(* PLC project EPEC_CU1.project, CODESYS V3.5 SP10 *)
(* stored: creationDateTime 2025-02-24T16:09:32.552285-06:00, modificationDateTime 2025-02-24T16:09:32.552285-06:00 *)

(* NOTE! NOTE! NOTE! NOTE! NOTE! NOTE! NOTE! NOTE! NOTE! NOTE! NOTE! This object is created by Epec MultiTool. User changes are overwritten when project is imported. Content: - EventCode channel IDs *)
{attribute 'qualified_only'}
{attribute 'strict'}
TYPE ChannelIDs : (Ch1 := 0, Ch2, Ch3, Ch4) BYTE;
END_TYPE

(* NOTE! NOTE! NOTE! NOTE! NOTE! NOTE! NOTE! NOTE! NOTE! NOTE! NOTE! This object is created by Epec MultiTool. User changes are overwritten when project is imported. Content: - EventCode device IDs *)
{attribute 'qualified_only'}
{attribute 'strict'}
TYPE DeviceIDs : (VoltageInput := 0, DigitalInput, CurrentInput, ParameterValidation) BYTE;
END_TYPE

TYPE IdentityObject : STRUCT
  VendorId : DWORD := 0;  (* Vendor ID *)
  ProductCode : DWORD := 0;  (* Product code *)
  Revision : DWORD := 0;  (* Revision number *)
  SerialNumber : DWORD := 0;  (* Serial number for control unit *)
END_STRUCT;
END_TYPE

VAR_GLOBAL CONSTANT  (* G_CONSTANTS - NOTE! NOTE! NOTE! NOTE! NOTE! NOTE! NOTE! NOTE! NOTE! NOTE! NOTE! This object is created by Epec MultiTool. User changes are overwritten when project is imported. Content: - Project specific constant definitions *)
  DIAG_TEMP_HIGH_LIMIT : DINT := 105;  (* Diagnostic limit constants *)
  DIAG_TEMP_LOW_LIMIT : DINT := -35;
  DIAG_TEMP_DELAY : UINT := 50;
  DIAG_SUPPLY_VOLTAGE_HIGH_LIMIT : DINT := 34000;
  DIAG_SUPPLY_VOLTAGE_LOW_LIMIT : DINT := 9000;
  DIAG_SUPPLY_VOLTAGE_DELAY : UINT := 95;
  DIAG_OUTPUT_GROUP1_HIGH_LIMIT : DINT := 34000;
  DIAG_OUTPUT_GROUP1_LOW_LIMIT : DINT := 9000;
  DIAG_OUTPUT_GROUP1_DELAY : UINT := 95;
  DIAG_5V_VAN_HIGH_LIMIT : DINT := 5250;
  DIAG_5V_VAN_LOW_LIMIT : DINT := 4750;
  DIAG_5V_VAN_DELAY : UINT := 50;
  DIAG_REF_DELAY : UINT := 50;
  DIAG_REF_TYPE_5V : BOOL := TRUE;  (* Reference output range selection [ TRUE = 5V, FALSE = 10V ] *)
  G_PARAMHANDLERKEYWORD : DWORD := 16#4EB1DA68;  (* Parameterhandler keyword *)
  G_PARAMETER_SAVE_STATUS_ERROR : BYTE := BYTE#16#00;
  G_PARAMETER_SAVE_STATUS_DONE : BYTE := BYTE#16#01;
  G_PARAMETER_SAVE_STATUS_IN_PROGRESS : BYTE := BYTE#16#FF;
  G_SAFE_PARAMETERS_AUTHENTICATED : BYTE := BYTE#1;
  G_SAFE_PARAMETERS_NOT_AUTHENTICATED : BYTE := BYTE#0;
END_VAR

{attribute 'qualified_only'}
VAR_GLOBAL  (* G_CAN - NOTE! NOTE! NOTE! NOTE! NOTE! NOTE! NOTE! NOTE! NOTE! NOTE! NOTE! This object is created by Epec MultiTool. User changes are overwritten when project is imported. Content: - CAN definitions *)
  Channel1 : EPEC_CANL2.Channel;
  Channel2 : EPEC_CANL2.Channel;
END_VAR

{attribute 'qualified_only'}
{attribute 'location' := '16#800'}
VAR_GLOBAL  (* G_Common *)
  ParHandler : EPEC_PH.ParameterHandler;  (* Parameterhandler. Utility library for ODSave. Library handles parameter image modification. *)
  ParameterArea : ARRAY[1..EPEC_HWD.LibParameters.G_PARAM_AREA_MAX_SIZE] OF BYTE;  (* Parameter image *)
  FastParHandler : EPEC_PH.ParameterHandler;
  FastParameterArea : ARRAY[1..EPEC_HWD.LibParameters.G_USER_VALUE_AREA_MAX_SIZE] OF BYTE;
  FastParameters : FastParameters;
  SaveFastParameters : BOOL := FALSE;
  ProjectKey : STRING(79) := '2JnCsjKPnmjYPqk';  (* Project key, used for validating the response code *)
END_VAR


{attribute 'qualified_only'}
{attribute 'location' := '16#800'}
VAR_GLOBAL  (* G_Logs *)
  ApplicationLog : EPEC_SERRLOG.ErrorLog;
  AppLogInitOK : BOOL;
END_VAR


{attribute 'qualified_only'}
{attribute 'location' := '16#800'}
VAR_GLOBAL  (* G_StatusFlags - NOTE! NOTE! NOTE! NOTE! NOTE! NOTE! NOTE! NOTE! NOTE! NOTE! NOTE! This object is created by Epec MultiTool. User changes are overwritten when project is imported. Content: - PLC_PRG status flags *)
  CANopenCan1NMTResetRequest : BOOL := FALSE;  (* Reset request flags tell if module is wanted to reset after current application cycle. *)
  CANopenCan2NMTResetRequest : BOOL := FALSE;
  SystemOk : BOOL := FALSE;
  CustomLEDControlEnable : BOOL := FALSE;  (* Flags to control the status LED from the application *)
  RedLED : BOOL := FALSE;
  GreenLED : BOOL := FALSE;
  BlueLED : BOOL := FALSE;
END_VAR

{attribute 'qualified_only'}
{attribute 'location' := '16#800'}
VAR_GLOBAL  (* G_SystemInfo - NOTE! NOTE! NOTE! NOTE! NOTE! NOTE! NOTE! NOTE! NOTE! NOTE! NOTE! This object is created by Epec MultiTool. User changes are overwritten when project is imported. Content: - System information common for all ODs. *)
  ProjectInfo : PROJECT_INFO;
  DeviceName : STRING(79);  (* 16#1008: Manufacturer device name *)
  HWVersion : STRING(79);  (* 16#1009: Manufacturer hardware version *)
  SWVersion : STRING(79);  (* 16#100A: Manufacturer software version *)
  Identity : IdentityObject;  (* 16#1018: Identity object *)
  ToolsVersion : ARRAY[1..1] OF DWORD;  (* 16#2030 Codesys version *)
  SoftwareInformation : ARRAY[1..10] OF STRING(79) := [''];  (* 16#2130 Software information Sub1: Application version Sub2: Additional version information Sub3: Reserved for future use Sub4: Reserved for future use Sub5: Reserved for future use Sub6: Reserved for future use Sub7: Reserved for future use Sub8: Reserved for future use Sub9: Reserved for future use Sub10: Reserved for future use *)
  CAN1_Comms : ARRAY[1..10] OF WORD := [10(0)];  (* 16#2150 CAN 1 Communication parameters Sub1: CODESYS communication enabled Sub2: CODESYS communication node-ID Sub3: Bit rate Sub4: Cable detection offset for CODESYS node-ID Sub5: Cable detection offset for PLCopen node-ID Sub6: Mask for cable detection pins Sub7: Reserved Sub8: Reserved Sub9: Reserved Sub10: PLCopen application node-ID in CAN1 *)
  CAN2_Comms : ARRAY[1..10] OF WORD := [10(0)];  (* 16#2151 CAN 2 Communication parameters Sub1: CODESYS communication enabled Sub2: CODESYS communication node-ID Sub3: Bit rate Sub4: Reserved Sub5: Reserved Sub6: Reserved Sub7: Reserved Sub8: Reserved Sub9: Reserved Sub10: PLCopen application node-ID in CAN2 *)
END_VAR

{attribute 'qualified_only'}
{attribute 'global_init_slot' := '49991'}
VAR_GLOBAL  (* G_CANopen_CAN1 - NOTE! NOTE! NOTE! NOTE! NOTE! NOTE! NOTE! NOTE! NOTE! NOTE! NOTE! This object is created by Epec MultiTool User changes are overwritten when project is imported Content - CANopen protocol variable definitions *)
  Device : EPEC_CANopen.Device;  (* CAN device *)
  OD : EPEC_CANopen.OD;  (* Object Dictionary data *)
  ODEntrys : ARRAY[1..70] OF EPEC_CANopen.ODEntry;
  Protocols : ARRAY[1..5] OF EPEC_CANopen.ProtocolEntry;  (* Protocol data *)
  HB : EPEC_CANopen.HBData;  (* Heartbeat producer/consumer protocol data *)
  HB_Handler : EPEC_CANopen.CANopenHB;  (* Heartbeat producer/consumer protocol handler *)
  NMT : EPEC_CANopen.NMTData;  (* NMT protocol data *)
  NMT_Handler : EPEC_CANopen.CANopenNMT;  (* NMT protocol handler *)
  SSDO : EPEC_CANopen.SSDOData;  (* SDO server protocol data *)
  SSDO_Handler : EPEC_CANopen.CANopenSDOServer;  (* SDO server protocol handler *)
  GFC : EPEC_CANopen.GFCData;  (* GFC protocol data *)
  GFC_Handler : EPEC_CANopen.CANopenGFC;  (* GFC protocol handler *)
  CSDOS : ARRAY[1..1] OF EPEC_CANopen.CANopenCSDO := [];  (* SDO client instances *)
  AppLogDomain : EPEC_CANopen.Domain;  (* 16#2171 Application log domain *)
  SaveAll : EPEC_ODSave.SaveODSaveAll;
  DeleteAll : EPEC_ODSave.SaveODDeleteAll;
  Initialize : EPEC_ODSave.SaveODInitialize;
  SaveData : ARRAY[0..3] OF EPEC_ODSave.SaveODSubIndexDescription := [(StartIndex := 16#1000, EndIndex := 16#FFFF, GroupNum := 1), (StartIndex := 16#1000, EndIndex := 16#1FFF, GroupNum := 1), (StartIndex := 16#2000, EndIndex := 16#FFFF, GroupNum := 1), (StartIndex := 16#0, EndIndex := 16#0, GroupNum := 1)];
  SaveSubData1010h : EPEC_ODSave.SaveODSubService;
END_VAR

{attribute 'qualified_only'}
{attribute 'location' := '16#800'}
{attribute 'global_init_slot' := '49990'}
VAR_GLOBAL  (* G_CANopen_CAN1_VAR - NOTE! NOTE! NOTE! NOTE! NOTE! NOTE! NOTE! NOTE! NOTE! NOTE! NOTE! This object is created by Epec MultiTool User changes are overwritten when project is imported Content - *)
  OD_Error : EPEC_CANopen.Errors := EPEC_CANopen.Errors.NotInitialized;
  ODSave_Error : EPEC_ODSave.SaveODErrors;
  Callback_Error : EPEC_CANopen.Errors := EPEC_CANopen.Errors.NotInitialized;
  ProtocolAdded : ARRAY[1..5] OF BOOL := [5(0)];
  HB_Error : EPEC_CANopen.Errors := EPEC_CANopen.Errors.NotInitialized;
  NMT_Error : EPEC_CANopen.Errors := EPEC_CANopen.Errors.NotInitialized;
  SSDO_Error : EPEC_CANopen.Errors := EPEC_CANopen.Errors.NotInitialized;
  GFC_Error : EPEC_CANopen.Errors := EPEC_CANopen.Errors.NotInitialized;
  GFC_Status : BYTE;  (* GFC status *)
  CSDO_Error : EPEC_CANopen.Errors := EPEC_CANopen.Errors.NotInitialized;
  SaveSigns1010 : ARRAY[0..3] OF DWORD;
END_VAR

{attribute 'qualified_only'}
{attribute 'location' := '16#800'}
VAR_GLOBAL  (* G_CAN1_VAR - NOTE! NOTE! NOTE! NOTE! NOTE! NOTE! NOTE! NOTE! NOTE! NOTE! NOTE! This object is created by Epec MultiTool User changes are overwritten when project is imported Content - CANopen OD index data *)
  DeviceType_Device1 : UDINT := 405;  (* 16#1000 Information about the device type *)
  ErrorReg_Device1 : USINT := 0;  (* 16#1001 Error information *)
  TPDO_DUMMY : BYTE := 0;  (* 16#2128 PDO Dummy Variable Index *)
  RPDO_DUMMY : BYTE := 0;  (* 16#2129 PDO Dummy Variable Index *)
  Parameter_CSV_unique_ID : UINT := 16#0000;  (* 16#2131 Parameter CSV unique ID *)
  ParameterSaveStatus : BYTE := 0;  (* 16#21FA Parameter save information *)
END_VAR

(* This PRG contains non safety-related code. The following attribute is autogenerated. Do not remove. *)
{attribute 'location' := '16#800'}
PROGRAM NVMemory
  VAR_INPUT
    i_Initialize : BOOL := TRUE;
  END_VAR
  VAR_OUTPUT
    o_InitReady : BOOL;
    o_InitError : BOOL;
    o_InputError : BOOL;
    o_ParameterBackupLoaded : BOOL;  (* Valid OD parameter backup image loaded during init. Note indication requires HWD lib 1.1.3.0. *)
    o_FastParameterBackupLoaded : BOOL;  (* Valid fast parameter backup image loaded during init. Note indication requires HWD lib 1.1.3.0. *)
    o_ODParameterError : EPEC_PH.ParamHandlerStatus := EPEC_PH.ParamHandlerStatus.NO_ERROR;
    o_FastParameterError : EPEC_PH.ParamHandlerStatus := EPEC_PH.ParamHandlerStatus.NO_ERROR;
    o_NVMemError : EPEC_SYSTEM.SYSTEM_ERROR_CODES := EPEC_SYSTEM.SYSTEM_ERROR_CODES.FW_ERR_OK;
    o_DM2Error : EPEC_PH.ParamHandlerStatus := EPEC_PH.ParamHandlerStatus.NO_ERROR;
    o_MachineTypeError : EPEC_PH.ParamHandlerStatus := EPEC_PH.ParamHandlerStatus.NO_ERROR;  (* Note indication requires HWD lib 1.1.5.0. *)
  END_VAR
  VAR
    parSaveBusy : BOOL := FALSE;
    parSaveDone : BOOL := FALSE;
    parSaveError : BOOL := FALSE;
    authenticated : BOOL := FALSE;
  END_VAR

            IF i_Initialize THEN
	EPEC_HWD.NVMem.SetParameterBackup(i_Enable := EPEC_HWD.LibParameters.G_PARAM_BACKUP_IN_USE);

	EPEC_HWD.NVMem.Init(
		i_NVMemoryIndex := 0,
		i_pParametersArea := ADR(G_Common.ParameterArea),
		i_ParameterAreaSize := SIZEOF(G_Common.ParameterArea),
		i_pParameterHandler := ADR(G_Common.ParHandler),
		i_pUserValuesArea := ADR(G_Common.FastParameterArea),
		i_UserValueAreaSize := SIZEOF(G_Common.FastParameterArea),
		i_pUserValueHandler := ADR(G_Common.FastParHandler),
		i_pUserValues := ADR(G_Common.FastParameters),
		i_UserValuesSize := SIZEOF(G_Common.FastParameters),
		i_pDM2Area := 0,
		i_DM2AreaSize := 0,
		i_pDM2Handler := 0,
		i_pMachineTypeArea := DWORD#0,
		i_MachineTypeAreaSize := UDINT#0,
		i_pMachineTypeHandler := DWORD#0,
		i_ParHandlerKeyword := G_CONSTANTS.G_PARAMHANDLERKEYWORD,
		o_InitReady => o_InitReady,
	);
	// Check if backup images were loaded during initialization
	IF o_InitReady THEN
		EPEC_HWD.NVMem.IsBackupLoaded(
			o_ParameterBackupLoaded => o_ParameterBackupLoaded,
			o_UserValueBackupLoaded => o_FastParameterBackupLoaded
		);
	END_IF
ELSE

	EPEC_HWD.NVMem(
		i_WriteParameters := G_Common.ParHandler.o_ParametersChanged,
		i_WriteUserValues := G_Common.SaveFastParameters,
		i_WriteDM2 := FALSE,
		i_WriteMachineType := FALSE,
		i_Authentication := authenticated,
		o_InitError => o_InitError,
		o_InputError => o_InputError,
		o_ParameterError => o_ODParameterError,
		o_UserValueError => o_FastParameterError,
		o_DM2Error => o_DM2Error,
		o_MachineTypeError => o_MachineTypeError,
		o_NVMemError => o_NVMemError,
		o_ParSaveBusy => parSaveBusy,
		o_ParSaveDone => parSaveDone,
		o_ParSaveError => parSaveError
	);

    (* Set parameter save status value *)
	IF parSaveBusy THEN
		G_CAN1_VAR.ParameterSaveStatus:= G_CONSTANTS.G_PARAMETER_SAVE_STATUS_IN_PROGRESS; 
	ELSIF parSaveDone THEN
		G_CAN1_VAR.ParameterSaveStatus:= G_CONSTANTS.G_PARAMETER_SAVE_STATUS_DONE; 
	ELSIF parSaveError THEN
		G_CAN1_VAR.ParameterSaveStatus:= G_CONSTANTS.G_PARAMETER_SAVE_STATUS_ERROR; 
	END_IF

	EPEC_SERRLOG.S_AddError_DWORD(i_ErrorCode:= ApplicationErrors.NVRAM_INIT, i_LibraryErrorCode:= BOOL_TO_DINT(o_InitError), i_Info1:= 0, i_Info2:= 0);
	EPEC_SERRLOG.S_AddError_DWORD(i_ErrorCode:= ApplicationErrors.NVRAM_INPUT, i_LibraryErrorCode:= BOOL_TO_DINT(o_InputError), i_Info1:= 0, i_Info2:= 0);
	EPEC_SERRLOG.S_AddError_DWORD(i_ErrorCode:= ApplicationErrors.NVRAM_FW, i_LibraryErrorCode:= o_NVMemError, i_Info1:= 0, i_Info2:= 0);
	EPEC_SERRLOG.S_AddError_DWORD(i_ErrorCode:= ApplicationErrors.NVRAM_OD, i_LibraryErrorCode:= INT_TO_DINT(o_ODParameterError), i_Info1:= 0, i_Info2:= 0);
	EPEC_SERRLOG.S_AddError_DWORD(i_ErrorCode:= ApplicationErrors.NVRAM_FASTPAR, i_LibraryErrorCode:= INT_TO_DINT(o_FastParameterError), i_Info1:= 0, i_Info2:= 0);
	EPEC_SERRLOG.S_AddError_DWORD(i_ErrorCode:= ApplicationErrors.NVRAM_MACHINETYPE, i_LibraryErrorCode:= INT_TO_DINT(o_MachineTypeError), i_Info1:= 0, i_Info2:= 0);


    (* User value save triggered, reset trigger *)
    G_Common.SaveFastParameters := FALSE;
END_IF
            
          
END_PROGRAM

(* Tool version : '8.1.9098.589' (MultiTool build version) Xml version : '1.0.10' (MultiTool xml file version) Control Unit : 'EPEC_CU1' (Name of the unit in MultiTool) Control Unit Type : 'EC44-020' (Type of the unit in MultiTool, including the functional version) CODESYS Profile : 'CODESYS V3.5 SP10' (CODESYS profile that was selected in MultiTool) Device Description Version: '3.5.13.67' (Device description version that was selected in MultiTool) Export Time : '24.02.2025 16:09.32' (Date and time when exported from MultiTool) Export Path : 'C:\Users\Pierre-Louis\Documents\02-UACH\1-Projets\1-Voltan\02-Réalisation\DEV\Projet_Voltan\Voltan_ECU\EPEC_CU1' (Path where MultiTool exported) Project File : 'C:\Users\Pierre-Louis\Documents\02-UACH\1-Projets\1-Voltan\02-Réalisation\DEV\Projet_Voltan\Voltan_ECU\Voltan_ECU.mtproject' (MultiTool project file name that was used) *)
{attribute 'location' := '16#800'}
PROGRAM PLC_PRG
  VAR_OUTPUT
    o_InitDone : BOOL := FALSE;
  END_VAR
  VAR
    ControlLED : EPEC_HWD.DiagnosticLED;
  END_VAR

            
// Initialize application log
IF NOT G_Logs.AppLogInitOK THEN
	G_Logs.AppLogInitOK := EPEC_SERRLOG.S_InitErrorLog(i_pErrorLog:= ADR(G_Logs.ApplicationLog));
END_IF

IF NOT o_InitDone AND G_Logs.AppLogInitOK THEN

    (* Code template non-safe FB initializations *)
    IF NOT Init_Entry.o_Ready THEN
        Init_Entry();
    ELSIF NOT Init_IO.o_Ready THEN
        Init_IO();
    ELSIF NOT EPEC_SHWD.S_EC44_Diagnostic.S_o_InitReady THEN
        EPEC_SHWD.S_EC44_Diagnostic.Init(
            S_i_SupplyVoltageHighLimit := G_CONSTANTS.DIAG_SUPPLY_VOLTAGE_HIGH_LIMIT,
            S_i_SupplyVoltageLowLimit := G_CONSTANTS.DIAG_SUPPLY_VOLTAGE_LOW_LIMIT,
            S_i_SupplyVoltageDiagDelay := G_CONSTANTS.DIAG_SUPPLY_VOLTAGE_DELAY,
            S_i_RefControlType5V := G_CONSTANTS.DIAG_REF_TYPE_5V,
            S_i_RefControlDiagDelay := G_CONSTANTS.DIAG_REF_DELAY,
            S_i_OutputGroup1HighVoltage := G_CONSTANTS.DIAG_OUTPUT_GROUP1_HIGH_LIMIT,
            S_i_OutputGroup1LowVoltage:= G_CONSTANTS.DIAG_OUTPUT_GROUP1_LOW_LIMIT,
            S_i_OutputGroup1DiagDelay:= G_CONSTANTS.DIAG_OUTPUT_GROUP1_DELAY,
            S_i_5VANHighVoltage:= G_CONSTANTS.DIAG_5V_VAN_HIGH_LIMIT,
            S_i_5VANLowVoltage:= G_CONSTANTS.DIAG_5V_VAN_LOW_LIMIT,
            S_i_5VANDiagDelay:= G_CONSTANTS.DIAG_5V_VAN_DELAY,
            S_i_TemperatureHighLimit:= G_CONSTANTS.DIAG_TEMP_HIGH_LIMIT,
            S_i_TemperatureLowLimit:= G_CONSTANTS.DIAG_TEMP_LOW_LIMIT,
            S_i_TemperatureDiagDelay:= G_CONSTANTS.DIAG_TEMP_DELAY);

    ELSIF NOT NVMemory.o_InitReady THEN
        NVMemory(i_Initialize:=TRUE);
	ELSIF NOT Inputs.o_InitReady THEN
		Inputs(i_Initialize:=TRUE);
	ELSIF NOT Init_CAN.o_Ready THEN
		Init_CAN();
	ELSIF NOT Init_CANopen_CAN1.o_Ready THEN
		Init_CANopen_CAN1();

    ELSE
        (* User non-safe initialization *)
        MainInit(o_MainInitReady=>o_InitDone);
    END_IF
ELSE
    (* Non-safe actions to execute before non-safe main program *)
	G_CAN.Channel1.CheckMessages();
	G_CAN.Channel2.CheckMessages();
	Inputs(i_Initialize:=FALSE);
	Handle_CANopen_CAN1();


    EPEC_SHWD.S_EC44_Diagnostic(
        i_RefChannel1  := Inputs.o_AI_REF_OUTPUT_MAIN_Diagnostic,
        i_SupplyVoltageInPin := Inputs.o_VIN_1_1_Diagnostic,
        i_SupplyBeforeSafetySwitch1 := Inputs.o_AI_POWER1_SUPPLY_Diagnostic,
        i_SupplyAfterSafetySwitch1  := Inputs.o_AI_POWER1_OUTPUT_Diagnostic,
        i_5VANChannel1 := Inputs.o_AI_5VAN_Diagnostic,
        i_PCBTemperatureChannel1 := Inputs.o_TEMP_PCB_MAIN_Diagnostic,
        i_PCBTemperatureChannel2 := Inputs.o_TEMP_PCB_RED_Diagnostic,
        i_MCUTemperature := Inputs.o_TEMP_MCU_Diagnostic,
        i_SBCTemperature := Inputs.o_AI_SBC_TEMP_Diagnostic
    );

	Handle_Diagnostic();

	// Read latest firmware errors to application log when FW is in error state
	IF EPEC_SHWD.S_EC44_Diagnostic.S_o_FWDiagnosticTaskStatus = EPEC_IODRV.DIAGNOSTIC_TASK_STATUS.EDiagnosticStatusError THEN
		Handle_Firmware_Errors(i_ReadErrors:= TRUE);
	END_IF


    (* User non-safe main program *)
    Main();

    (* Non-safe actions to execute after non-safe main program *)

    NVMemory(i_Initialize:=FALSE);

    (* Boot application if NMT reset requested *)
    IF G_StatusFlags.CANopenCan1NMTResetRequest OR G_StatusFlags.CANopenCan2NMTResetRequest THEN
        EPEC_SYSTEM.BOOT_APPLICATION_KILL_RTS();
    END_IF
END_IF

ControlLED(
    i_InitState := NOT PLC_PRG.o_Initdone,
    i_ApplicationInSafeState := NOT EPEC_SHWD.S_EC44_Diagnostic.S_o_OutputGroup1Control,
    i_SystemOk := G_StatusFlags.SystemOk,
    i_CustomLEDControl := G_StatusFlags.CustomLEDControlEnable,
    i_RedLED := G_StatusFlags.RedLED,
    i_GreenLED := G_StatusFlags.GreenLED,
    i_BlueLED := G_StatusFlags.BlueLED,
    o_Error =>
);


              
          
END_PROGRAM

(* NOTE! NOTE! NOTE! NOTE! NOTE! NOTE! NOTE! NOTE! NOTE! NOTE! NOTE! This object is created by Epec MultiTool User changes are overwritten when project is imported Content - Initialization of CAN channels This PRG contains non safety-related code. The following attribute is autogenerated. Do not remove. *)
{attribute 'location' := '16#800'}
PROGRAM Init_CAN
  VAR_OUTPUT
    o_Ready : BOOL := FALSE;
    o_Error : BOOL := FALSE;
    o_CAN1InitError : EPEC_CANVXD.ERROR := EPEC_CANVXD.ERROR.CHANNEL_NOT_INITIALIZED;
    o_CAN2InitError : EPEC_CANVXD.ERROR := EPEC_CANVXD.ERROR.CHANNEL_NOT_INITIALIZED;
  END_VAR

            o_CAN1InitError := G_CAN.Channel1.InitCAN(i_Channel := 0, i_BitRate := G_SystemInfo.CAN1_Comms[3], i_Flags := 0);
o_CAN2InitError := G_CAN.Channel2.InitCAN(i_Channel := 1, i_BitRate := EPEC_CANVXD.BITRATE_250K, i_Flags := 0);

IF EPEC_CANVXD.ERROR.NO_ERROR = o_CAN1InitError AND
	EPEC_CANVXD.ERROR.NO_ERROR = o_CAN2InitError THEN
	o_Error := FALSE;
ELSE
	o_Error := TRUE;

	EPEC_SERRLOG.S_AddError_DWORD(i_ErrorCode:= ApplicationErrors.CAN_INIT, i_LibraryErrorCode:= INT_TO_DINT(o_CAN1InitError), i_Info1:= 0, i_Info2:= 1);
	EPEC_SERRLOG.S_AddError_DWORD(i_ErrorCode:= ApplicationErrors.CAN_INIT, i_LibraryErrorCode:= INT_TO_DINT(o_CAN2InitError), i_Info1:= 0, i_Info2:= 2);
END_IF

o_Ready := TRUE;

          
END_PROGRAM

(* NOTE! NOTE! NOTE! NOTE! NOTE! NOTE! NOTE! NOTE! NOTE! NOTE! NOTE! This object is created by Epec MultiTool User changes are overwritten when project is imported Content - Set system information common for all ODs. This PRG contains non safety-related code. The following attribute is autogenerated. Do not remove. *)
{attribute 'location' := '16#800'}
PROGRAM Init_Entry
  VAR_OUTPUT
    o_Ready : BOOL;
  END_VAR
  VAR
    Can2NodeId : WORD;
    Can2PLCopenNodeId : WORD;
    Can2BitRate : WORD;
    ReadBytes : DWORD;
    RandomNumber : UDINT;
    SystemParameters : EPEC_HW.SystemParameters;
  END_VAR

            SystemParameters.ReadData();

/// 16#1008: Manufacturer device name
EPEC_SYSTEM.SystemParametersRead (16#1008,0,79,ADR(G_SystemInfo.DeviceName),ADR(ReadBytes));
 /// 16#1009: Manufacturer hardware version
EPEC_SYSTEM.SystemParametersRead (16#1009,0,79,ADR(G_SystemInfo.HWVersion),ADR(ReadBytes));
/// 16#100A: Manufacturer software version
G_SystemInfo.SWVersion := SystemParameters.o_SoftwareVersion;
/// 16#1018: Identity object 
G_SystemInfo.Identity.VendorId := SystemParameters.o_VendorId;          /// Vendor ID
G_SystemInfo.Identity.ProductCode := SystemParameters.o_ProductCode;    /// Product code
G_SystemInfo.Identity.Revision := SystemParameters.o_RevisionNumber;    /// Revision number
G_SystemInfo.Identity.SerialNumber := SystemParameters.o_SerialNumber;  /// Serial number for control unit
/// 16#2030 Codesys version
G_SystemInfo.ToolsVersion[1] := DWORD#50659328;
/// 16#2150 CAN 1 Communication parameters
G_SystemInfo.CAN1_Comms := SystemParameters.i_CAN1;

/// Read parameters for CAN2 from firmware
EPEC_SYSTEM.SystemParametersRead (16#2151,2,2,ADR(Can2NodeId),ADR(ReadBytes));
EPEC_SYSTEM.SystemParametersRead (16#2151,3,2,ADR(Can2BitRate),ADR(ReadBytes));
EPEC_SYSTEM.SystemParametersRead (16#2151,10,2,ADR(Can2PLCopenNodeId),ADR(ReadBytes));

/// Set variables to communication arrays 
G_SystemInfo.CAN2_Comms[2] := Can2NodeId;
G_SystemInfo.CAN2_Comms[3] := Can2BitRate;
G_SystemInfo.CAN2_Comms[10] := Can2PLCopenNodeId;

o_Ready:= TRUE;

          
END_PROGRAM

(* NOTE! NOTE! NOTE! NOTE! NOTE! NOTE! NOTE! NOTE! NOTE! NOTE! NOTE! This object is created by Epec MultiTool User changes are overwritten when project is imported Content - Non-safe system status update This PRG contains non safety-related code. The following attribute is autogenerated. Do not remove. *)
{attribute 'location' := '16#800'}
PROGRAM Handle_Diagnostic

            (* System Ok conditions *)
G_StatusFlags.SystemOk:=
		EPEC_SHWD.S_EC44_Diagnostic.S_o_DiagStatusOk AND			(* System diagnostic ok *)
		NOT Init_CAN.o_Error AND			(* No errors in bus init *)
		NOT Init_CANopen_CAN1.o_Error;


// Check HW diagnostic errors when diagnostic is enabled
IF EPEC_SHWD.S_EC44_Diagnostic.S_o_Running AND NOT EPEC_SHWD.S_EC44_Diagnostic.S_o_DiagStatusOk THEN
	EPEC_SERRLOG.S_AddError_DWORD(
		i_ErrorCode := ApplicationErrors.HW_DIAGNOSTIC_FAULT,
		i_LibraryErrorCode := EPEC_SERRLOG.LibConstants.G_ErrorNA,
		i_Info1 := 0,
		i_Info2 := 0);

	// output group 1
	EPEC_SERRLOG.S_AddError_BYTE(
		i_ErrorCode := ApplicationErrors.HW_DIAG_OUT_PWR_GRP_1,
		i_LibraryErrorCode := EPEC_SHWD.S_EC44_Diagnostic.o_OutputGroup1Control_EC.EventID,
		i_Info1 := EPEC_SHWD.S_EC44_Diagnostic.o_OutputGroup1Control_EC.FunctionID,
		i_Info2 := EPEC_SHWD.S_EC44_Diagnostic.o_OutputGroup1Control_EC.DeviceID,
		i_Info3 := EPEC_SHWD.S_EC44_Diagnostic.o_OutputGroup1Control_EC.ChannelID,
		i_Info4 := 0,
		i_Info5 := 0,
		i_Info6 := 0,
		i_Info7 := 0,
		i_Info8 := 0);

	// REF output
	EPEC_SERRLOG.S_AddError_BYTE(
		i_ErrorCode := ApplicationErrors.HW_DIAG_OUT_REF_1,
		i_LibraryErrorCode := EPEC_SHWD.S_EC44_Diagnostic.o_RefControl_EC.EventID,
		i_Info1 := EPEC_SHWD.S_EC44_Diagnostic.o_RefControl_EC.FunctionID,
		i_Info2 := EPEC_SHWD.S_EC44_Diagnostic.o_RefControl_EC.DeviceID,
		i_Info3 := EPEC_SHWD.S_EC44_Diagnostic.o_RefControl_EC.ChannelID,
		i_Info4 := 0,
		i_Info5 := 0,
		i_Info6 := 0,
		i_Info7 := 0,
		i_Info8 := 0);

	// supply voltage
	EPEC_SERRLOG.S_AddError_BYTE(
		i_ErrorCode := ApplicationErrors.HW_DIAG_IN_SUPPLY,
		i_LibraryErrorCode := EPEC_SHWD.S_EC44_Diagnostic.o_SupplyVoltag_EC.EventID,
		i_Info1 := EPEC_SHWD.S_EC44_Diagnostic.o_SupplyVoltag_EC.FunctionID,
		i_Info2 := EPEC_SHWD.S_EC44_Diagnostic.o_SupplyVoltag_EC.DeviceID,
		i_Info3 := EPEC_SHWD.S_EC44_Diagnostic.o_SupplyVoltag_EC.ChannelID,
		i_Info4 := 0,
		i_Info5 := 0,
		i_Info6 := 0,
		i_Info7 := 0,
		i_Info8 := 0);

	// 5VAN
	EPEC_SERRLOG.S_AddError_BYTE(
		i_ErrorCode := ApplicationErrors.HW_DIAG_IN_5VAN,
		i_LibraryErrorCode := EPEC_SHWD.S_EC44_Diagnostic.o_5VAN_EC.EventID,
		i_Info1 := EPEC_SHWD.S_EC44_Diagnostic.o_5VAN_EC.FunctionID,
		i_Info2 := EPEC_SHWD.S_EC44_Diagnostic.o_5VAN_EC.DeviceID,
		i_Info3 := EPEC_SHWD.S_EC44_Diagnostic.o_5VAN_EC.ChannelID,
		i_Info4 := 0,
		i_Info5 := 0,
		i_Info6 := 0,
		i_Info7 := 0,
		i_Info8 := 0);

	// MCU temperature
	EPEC_SERRLOG.S_AddError_BYTE(
		i_ErrorCode := ApplicationErrors.HW_DIAG_IN_MCU_TEMP,
		i_LibraryErrorCode := EPEC_SHWD.S_EC44_Diagnostic.o_MCUTemperatureEC.EventID,
		i_Info1 := EPEC_SHWD.S_EC44_Diagnostic.o_MCUTemperatureEC.FunctionID,
		i_Info2 := EPEC_SHWD.S_EC44_Diagnostic.o_MCUTemperatureEC.DeviceID,
		i_Info3 := EPEC_SHWD.S_EC44_Diagnostic.o_MCUTemperatureEC.ChannelID,
		i_Info4 := 0,
		i_Info5 := 0,
		i_Info6 := 0,
		i_Info7 := 0,
		i_Info8 := 0);

	// SBC temperature
	EPEC_SERRLOG.S_AddError_BYTE(
		i_ErrorCode := ApplicationErrors.HW_DIAG_IN_SBC_TEMP,
		i_LibraryErrorCode := EPEC_SHWD.S_EC44_Diagnostic.o_SBCTemperatureEC.EventID,
		i_Info1 := EPEC_SHWD.S_EC44_Diagnostic.o_SBCTemperatureEC.FunctionID,
		i_Info2 := EPEC_SHWD.S_EC44_Diagnostic.o_SBCTemperatureEC.DeviceID,
		i_Info3 := EPEC_SHWD.S_EC44_Diagnostic.o_SBCTemperatureEC.ChannelID,
		i_Info4 := 0,
		i_Info5 := 0,
		i_Info6 := 0,
		i_Info7 := 0,
		i_Info8 := 0);

	// PCB temperature 1
	EPEC_SERRLOG.S_AddError_BYTE(
		i_ErrorCode := ApplicationErrors.HW_DIAG_IN_PCB_TEMP_1,
		i_LibraryErrorCode := EPEC_SHWD.S_EC44_Diagnostic.o_PCBTemperatureCh1_EC.EventID,
		i_Info1 := EPEC_SHWD.S_EC44_Diagnostic.o_PCBTemperatureCh1_EC.FunctionID,
		i_Info2 := EPEC_SHWD.S_EC44_Diagnostic.o_PCBTemperatureCh1_EC.DeviceID,
		i_Info3 := EPEC_SHWD.S_EC44_Diagnostic.o_PCBTemperatureCh1_EC.ChannelID,
		i_Info4 := 0,
		i_Info5 := 0,
		i_Info6 := 0,
		i_Info7 := 0,
		i_Info8 := 0);

	// PCB temperature 2
	EPEC_SERRLOG.S_AddError_BYTE(
		i_ErrorCode := ApplicationErrors.HW_DIAG_IN_PCB_TEMP_2,
		i_LibraryErrorCode := EPEC_SHWD.S_EC44_Diagnostic.o_PCBTemperatureCh2_EC.EventID,
		i_Info1 := EPEC_SHWD.S_EC44_Diagnostic.o_PCBTemperatureCh2_EC.FunctionID,
		i_Info2 := EPEC_SHWD.S_EC44_Diagnostic.o_PCBTemperatureCh2_EC.DeviceID,
		i_Info3 := EPEC_SHWD.S_EC44_Diagnostic.o_PCBTemperatureCh2_EC.ChannelID,
		i_Info4 := 0,
		i_Info5 := 0,
		i_Info6 := 0,
		i_Info7 := 0,
		i_Info8 := 0);

END_IF



          
END_PROGRAM

(* NOTE! NOTE! NOTE! NOTE! NOTE! NOTE! NOTE! NOTE! NOTE! NOTE! NOTE! This object is created by Epec MultiTool User changes are overwritten when project is imported Content - Reads firmware error codes to application error log This PRG contains non safety-related code. The following attribute is autogenerated. Do not remove. *)
{attribute 'location' := '16#800'}
PROGRAM Handle_Firmware_Errors
  VAR_INPUT
    i_ReadErrors : BOOL;
  END_VAR
  VAR
    readErrorsOld : BOOL;
    fw_entries : ARRAY [1..EPEC_SERRLOG.LibParameters.G_ERROR_LOG_MAX_LINES] OF EPEC_SYSTEM.SystemLogEntry;
    return_code : EPEC_SYSTEM.SYSTEM_ERROR_CODES;
    lines_found : UDINT;
    i : UDINT;
    previous_time : UDINT;
    boot_detected : BOOL;
    fw_log_startupid : UDINT := UDINT#0;
    fw_log_startupid_exist : BOOL := FALSE;
    fw_log_startupid_size : DWORD;
  END_VAR

            IF i_ReadErrors AND NOT readErrorsOld THEN
	// Read FW log startup id value, if supported by FW
	return_code := EPEC_SYSTEM.SystemParametersRead(i_Index:=16#2039, i_SubIndex:=2, i_pBufferSize:=SIZEOF(fw_log_startupid), i_pBuffer:=ADR(fw_log_startupid), i_pNbrOfReadByte:=ADR(fw_log_startupid_size));

	// Check if read was success
	IF return_code = EPEC_SYSTEM.SYSTEM_ERROR_CODES.FW_ERR_OK THEN
		fw_log_startupid_exist := TRUE;
	ELSE
		fw_log_startupid_exist := FALSE;
	END_IF

	// Read firmware errors
	return_code:= EPEC_SYSTEM.GetFWLogTail(
		i_Count:= EPEC_SERRLOG.LibParameters.G_ERROR_LOG_MAX_LINES,
		i_logEntryArray:= ADR(fw_entries),
		o_Found => lines_found
	);

	IF return_code = EPEC_SYSTEM.SYSTEM_ERROR_CODES.FW_ERR_OK AND lines_found > UDINT#0 THEN
		// Check if startup id is supported by FW
		IF fw_log_startupid_exist THEN
			// Add errors from buffer until startup id is found 
			FOR i:= 1 TO EPEC_SERRLOG.LibParameters.G_ERROR_LOG_MAX_LINES DO
				IF i <= lines_found AND fw_entries[i].Identifier >= fw_log_startupid THEN
					S_AddError_DWORD(
						i_ErrorCode:= ApplicationErrors.FW_ERROR,
						i_LibraryErrorCode:= fw_entries[i].Error,
						i_Info1:= fw_entries[i].Info,
						i_Info2:= fw_entries[i].Identifier);
				END_IF
			END_FOR
		ELSE
			// Add first error
			S_AddError_DWORD(
				i_ErrorCode:= ApplicationErrors.FW_ERROR,
				i_LibraryErrorCode:= fw_entries[1].Error,
				i_Info1:= fw_entries[1].Info,
				i_Info2:= fw_entries[1].Identifier);

			previous_time:= fw_entries[1].Timestamp;
			boot_detected:= FALSE;

			// Add errors until timestamp rollover is detected
			FOR i:= 2 TO EPEC_SERRLOG.LibParameters.G_ERROR_LOG_MAX_LINES DO
				IF i <= lines_found AND fw_entries[i].Timestamp <= previous_time AND NOT boot_detected THEN
					S_AddError_DWORD(
						i_ErrorCode:= ApplicationErrors.FW_ERROR,
						i_LibraryErrorCode:= fw_entries[i].Error,
						i_Info1:= fw_entries[i].Info,
						i_Info2:= fw_entries[i].Identifier);

					previous_time:= fw_entries[i].Timestamp;

				ELSIF fw_entries[i].Timestamp > previous_time THEN
					boot_detected := TRUE;
				END_IF
			END_FOR
		END_IF
	END_IF
END_IF
readErrorsOld:= i_ReadErrors;

          
END_PROGRAM

(* NOTE! NOTE! NOTE! NOTE! NOTE! NOTE! NOTE! NOTE! NOTE! NOTE! NOTE! This object is created by Epec MultiTool User changes are overwritten when project is imported Content - CANopen initialization - Includes Init_CANopen_OD1 - CANopen data update This PRG contains non safety-related code. The following attribute is autogenerated. Do not remove. *)
{attribute 'location' := '16#800'}
PROGRAM Init_CANopen_CAN1
  VAR_OUTPUT
    o_Ready : BOOL := FALSE;
    o_Error : BOOL := FALSE;
  END_VAR

            G_CANopen_CAN1.Device.itfCanChannel:=G_CAN.Channel1; (*Connect device to can channel*)
G_CANopen_CAN1.Device.NodeID := BYTE#1;
G_CANopen_CAN1.NMT.NmtState:=EPEC_CANopen.NMTState.BootUp; (* Set NMT status to BOOTUP *)

(*Initialize OD's data structures*)
G_CANopen_CAN1.OD.EntryCount:=SIZEOF(G_CANopen_CAN1.ODEntrys)/SIZEOF(G_CANopen_CAN1.ODEntrys[1]); (*Max entries of given OD(CANopenDeviceODEntrys array)*)
G_CANopen_CAN1.OD.InOrder:=FALSE; (*OD isn't in order*)
G_CANopen_CAN1.OD.NextFree:=0; (*OD does not have any entries yet*)
G_CANopen_CAN1.OD.pODEntry:=ADR(G_CANopen_CAN1.ODEntrys); (*Pointer to OD array*)

(*Define NMT protocol*)
G_CANopen_CAN1.Protocols[1].Protocol:=EPEC_CANopen.ProtocolType.NMT;
G_CANopen_CAN1.Protocols[1].pData:=ADR(G_CANopen_CAN1.NMT);
G_CANopen_CAN1.Protocols[1].itfProtocol:=G_CANopen_CAN1.NMT_Handler;
G_CANopen_CAN1.Protocols[1].pError:=ADR(G_CANopen_CAN1_VAR.NMT_Error);
G_CANopen_CAN1_VAR.ProtocolAdded[1] := CANopenDeviceAddProtocol( (* Add to protocol stack *)
	i_pDevice:=ADR(G_CANopen_CAN1.Device),
	i_pProtocol:=ADR(G_CANopen_CAN1.Protocols[1]),
);

(*Initialize NMT protocol*)
IF G_CANopen_CAN1_VAR.ProtocolAdded[1] THEN
	G_CANopen_CAN1.NMT_Handler.Init(
		i_pDevice := ADR(G_CANopen_CAN1.Device),
		i_ThisIsMaster := FALSE,
		i_StartInterval :=  1000,
		i_pMonitoredNodes := 0,
		i_NumberOfNodes := 0,
		i_SimultaneousSlaveConfiguration := FALSE,
		o_Error => G_CANopen_CAN1_VAR.NMT_Error
	);
ELSE
	G_CANopen_CAN1_VAR.NMT_Error := EPEC_CANopen.Errors.ProtocolDataMissing;
END_IF

(*Define OD protocol*)
G_CANopen_CAN1.Protocols[2].Protocol:=EPEC_CANopen.ProtocolType.OD;
G_CANopen_CAN1.Protocols[2].pData:=ADR(G_CANopen_CAN1.OD);
G_CANopen_CAN1.Protocols[2].pError:=ADR(G_CANopen_CAN1_VAR.OD_Error);
G_CANopen_CAN1_VAR.ProtocolAdded[2] := CANopenDeviceAddProtocol( (* Add to protocol stack *)
	i_pDevice:=ADR(G_CANopen_CAN1.Device),
	i_pProtocol:=ADR(G_CANopen_CAN1.Protocols[2]),
);
IF NOT G_CANopen_CAN1_VAR.ProtocolAdded[2] THEN
	G_CANopen_CAN1_VAR.OD_Error := EPEC_CANopen.Errors.ProtocolDataMissing;
END_IF

(*Define HB protocol
- Uses NMT and OD protocol data, thus need to be defined after them.
*)
G_CANopen_CAN1.HB.HeartBeat.PT := T#200MS; (* HB producer time *)

G_CANopen_CAN1.Protocols[3].Protocol:=EPEC_CANopen.ProtocolType.HB;
G_CANopen_CAN1.Protocols[3].pData:=ADR(G_CANopen_CAN1.HB);
G_CANopen_CAN1.Protocols[3].itfProtocol:=G_CANopen_CAN1.HB_Handler;
G_CANopen_CAN1.Protocols[3].pError:=ADR(G_CANopen_CAN1_VAR.HB_Error);
G_CANopen_CAN1_VAR.ProtocolAdded[3] := CANopenDeviceAddProtocol( (* Add to protocol stack *)
	i_pDevice:=ADR(G_CANopen_CAN1.Device),
	i_pProtocol:=ADR(G_CANopen_CAN1.Protocols[3]),
);

(* Initialize HB protocol *)
IF G_CANopen_CAN1_VAR.ProtocolAdded[3] THEN

	(* Add monitored nodes *)
	G_CANopen_CAN1.HB_Handler.Init(
		i_pDevice := ADR(G_CANopen_CAN1.Device),
		o_Error => G_CANopen_CAN1_VAR.HB_Error
	);
ELSE
	G_CANopen_CAN1_VAR.HB_Error := EPEC_CANopen.Errors.ProtocolDataMissing;
END_IF

(*Define SSDO protocol*)
G_CANopen_CAN1.Protocols[4].Protocol:=EPEC_CANopen.ProtocolType.SSDO;
G_CANopen_CAN1.Protocols[4].pData:=ADR(G_CANopen_CAN1.SSDO);
G_CANopen_CAN1.Protocols[4].itfProtocol:=G_CANopen_CAN1.SSDO_Handler;
G_CANopen_CAN1.Protocols[4].pError:=ADR(G_CANopen_CAN1_VAR.SSDO_Error);
G_CANopen_CAN1_VAR.ProtocolAdded[4] := CANopenDeviceAddProtocol( (* Add to protocol stack *)
	i_pDevice:=ADR(G_CANopen_CAN1.Device),
	i_pProtocol:=ADR(G_CANopen_CAN1.Protocols[4])
);
IF G_CANopen_CAN1_VAR.ProtocolAdded[4] THEN
	G_CANopen_CAN1.SSDO_Handler.Init(
		i_pDevice := ADR(G_CANopen_CAN1.Device),
		o_Error => G_CANopen_CAN1_VAR.SSDO_Error
	);
ELSE
	G_CANopen_CAN1_VAR.SSDO_Error := EPEC_CANopen.Errors.ProtocolDataMissing;
END_IF

(*Define GFC protocol*)
G_CANopen_CAN1.Protocols[5].Protocol:=EPEC_CANopen.ProtocolType.GFC;
G_CANopen_CAN1.Protocols[5].pData:=ADR(G_CANopen_CAN1.GFC);
G_CANopen_CAN1.Protocols[5].itfProtocol:=G_CANopen_CAN1.GFC_Handler;
G_CANopen_CAN1.Protocols[5].pError:=ADR(G_CANopen_CAN1_VAR.GFC_Error);
G_CANopen_CAN1_VAR.ProtocolAdded[5] := CANopenDeviceAddProtocol(  (* Add to protocol stack *)
	i_pDevice:=ADR(G_CANopen_CAN1.Device),
	i_pProtocol:=ADR(G_CANopen_CAN1.Protocols[5])
);
IF G_CANopen_CAN1_VAR.ProtocolAdded[5] THEN
	G_CANopen_CAN1.GFC_Handler.Init(
		i_pDevice := ADR(G_CANopen_CAN1.Device),
		i_pStatus:=ADR(G_CANopen_CAN1_VAR.GFC_Status),
		o_Error => G_CANopen_CAN1_VAR.GFC_Error
	);
ELSE
	G_CANopen_CAN1_VAR.GFC_Error := EPEC_CANopen.Errors.ProtocolDataMissing;
END_IF

(* Init CSDO instance array for bus *)
EPEC_CANopen.CANopenSDOManager.Init(
	i_pDevice:=ADR(G_CANopen_CAN1.Device),
	i_pCsdoArrayStart:=ADR(G_CANopen_CAN1.CSDOS),
	i_CsdoArraySize:=SIZEOF(G_CANopen_CAN1.CSDOS)/SIZEOF(G_CANopen_CAN1.CSDOS[1]),
	o_Error=>G_CANopen_CAN1_VAR.CSDO_Error
);

(* Add index data to OD *)
Init_CANopen_OD1(); (* Must be done before initing PDOs and SRDOs. *)

(*Initialize OD save*)
G_CANopen_CAN1.SaveAll.Init(i_pParamHandler:=ADR(G_Common.ParHandler));
G_CANopen_CAN1.DeleteAll.Init(i_pParamHandler:=ADR(G_Common.ParHandler));
G_CANopen_CAN1.SaveSubData1010h.pSaveSigns := ADR(G_CANopen_CAN1_VAR.SaveSigns1010[0]);
G_CANopen_CAN1.SaveSubData1010h.NumOfEntrys := 4;
G_CANopen_CAN1.SaveSubData1010h.pSaveIndexData := ADR(G_CANopen_CAN1.SaveData[0]);
G_CANopen_CAN1.SaveData[3].itfSaveAll := G_CANopen_CAN1.SaveAll;
G_CANopen_CAN1.SaveData[3].itfDeleteAll := G_CANopen_CAN1.DeleteAll;
G_CANopen_CAN1.OD.pAdditionalData := ADR(G_CANopen_CAN1.SaveSubData1010h);

IF G_CANopen_CAN1_VAR.OD_Error = EPEC_CANopen.Errors.NoError THEN
	G_CANopen_CAN1.Initialize(i_pOD:=ADR(G_CANopen_CAN1.OD), i_pParamHandler:=ADR(G_Common.ParHandler), o_Error => G_CANopen_CAN1_VAR.ODSave_Error);
END_IF

(* Check all protocol init status flags *)
IF G_CANopen_CAN1_VAR.NMT_Error = EPEC_CANopen.Errors.NoError AND
	G_CANopen_CAN1_VAR.SSDO_Error = EPEC_CANopen.Errors.NoError AND
	G_CANopen_CAN1_VAR.OD_Error = EPEC_CANopen.Errors.NoError AND
	G_CANopen_CAN1_VAR.HB_Error = EPEC_CANopen.Errors.NoError AND
	G_CANopen_CAN1_VAR.CSDO_Error = EPEC_CANopen.Errors.NoError AND
	G_CANopen_CAN1_VAR.GFC_Error = EPEC_CANopen.Errors.NoError
THEN
	o_Error := FALSE; (* No errors in protocol inits *)
ELSE
	o_Error := TRUE;

	EPEC_SERRLOG.S_AddError_DWORD(i_ErrorCode:= ApplicationErrors.CANOPEN_INIT_NMT, i_LibraryErrorCode:= INT_TO_DINT(G_CANopen_CAN1_VAR.NMT_Error), i_Info1:= 0, i_Info2:= 1);
	EPEC_SERRLOG.S_AddError_DWORD(i_ErrorCode:= ApplicationErrors.CANOPEN_INIT_SSDO, i_LibraryErrorCode:= INT_TO_DINT(G_CANopen_CAN1_VAR.SSDO_Error), i_Info1:= 0, i_Info2:= 1);
	EPEC_SERRLOG.S_AddError_DWORD(i_ErrorCode:= ApplicationErrors.CANOPEN_INIT_OD, i_LibraryErrorCode:= INT_TO_DINT(G_CANopen_CAN1_VAR.OD_Error), i_Info1:= 0, i_Info2:= 1);
	EPEC_SERRLOG.S_AddError_DWORD(i_ErrorCode:= ApplicationErrors.CANOPEN_INIT_HB, i_LibraryErrorCode:= INT_TO_DINT(G_CANopen_CAN1_VAR.HB_Error), i_Info1:= 0, i_Info2:= 1);
	EPEC_SERRLOG.S_AddError_DWORD(i_ErrorCode:= ApplicationErrors.CANOPEN_INIT_CSDO, i_LibraryErrorCode:= INT_TO_DINT(G_CANopen_CAN1_VAR.CSDO_Error), i_Info1:= 0, i_Info2:= 1);
	EPEC_SERRLOG.S_AddError_DWORD(i_ErrorCode:= ApplicationErrors.CANOPEN_INIT_GFC, i_LibraryErrorCode:= INT_TO_DINT(G_CANopen_CAN1_VAR.GFC_Error), i_Info1:= 0, i_Info2:= 1);

END_IF

o_Ready:=TRUE;

          
END_PROGRAM

(* NOTE! NOTE! NOTE! NOTE! NOTE! NOTE! NOTE! NOTE! NOTE! NOTE! NOTE! This object is created by Epec MultiTool User changes are overwritten when project is imported Content - CANopen object dictionary initialization This PRG contains non safety-related code. The following attribute is autogenerated. Do not remove. *)
{attribute 'location' := '16#800'}
PROGRAM Init_CANopen_OD1

            (*16#0001..16#0009 Default types *)
G_CANopen_CAN1_VAR.OD_Error := EPEC_CANopen.CANopenODAddDefautTypes(
	i_pOD:= ADR(G_CANopen_CAN1.OD)
);

(* 16#1000 Information about the device type *)
IF G_CANopen_CAN1_VAR.OD_Error = EPEC_CANopen.Errors.NoError THEN
	G_CANopen_CAN1_VAR.OD_Error := CANopenODAddLine(
		i_pOD := ADR(G_CANopen_CAN1.OD),(*Address of Object dictionary where index will be added*)
		i_Index := G_CANOPEN_ODINDEX_DEVICE_TYPE,
		i_ObjectCode := EPEC_CANopen.ObjectCode.OD_VAR,(*Type of index*)
		i_NumOfSubids := USINT#0,(*Number of subindexes*)
		i_TypeSpec := EPEC_CANopen.DataType.Deftype_UNSIGNED32,(*Index datatype, either user defined or standard CiA 301*)
		i_ObjectAccess := G_CANOPEN_OD_ACCESS_NOWRITE OR G_CANOPEN_OD_ACCESS_SUB0NOWRITE,
		i_Sub0data := USINT#0,(*Value of subindex0 in array or (def)struct*)
		i_pIndexData := ADR(G_CAN1_VAR.DeviceType_Device1),
		i_itfSDOHandler := DWORD#0
	);
END_IF

(* 16#1001 Error information *)
IF G_CANopen_CAN1_VAR.OD_Error = EPEC_CANopen.Errors.NoError THEN
	G_CANopen_CAN1_VAR.OD_Error := CANopenODAddLine(
		i_pOD := ADR(G_CANopen_CAN1.OD),(*Address of Object dictionary where index will be added*)
		i_Index := G_CANOPEN_ODINDEX_ERROR_REGISTER,
		i_ObjectCode := EPEC_CANopen.ObjectCode.OD_VAR,(*Type of index*)
		i_NumOfSubids := USINT#0,(*Number of subindexes*)
		i_TypeSpec := EPEC_CANopen.DataType.Deftype_UNSIGNED8,(*Index datatype, either user defined or standard CiA 301*)
		i_ObjectAccess := G_CANOPEN_OD_ACCESS_NOWRITE OR G_CANOPEN_OD_ACCESS_SUB0NOWRITE,
		i_Sub0data := USINT#0,(*Value of subindex0 in array or (def)struct*)
		i_pIndexData := ADR(G_CAN1_VAR.ErrorReg_Device1),
		i_itfSDOHandler := DWORD#0
	);
END_IF

(* 16#1008 Manufacturer device name *)
IF G_CANopen_CAN1_VAR.OD_Error = EPEC_CANopen.Errors.NoError THEN
	G_CANopen_CAN1_VAR.OD_Error := CANopenODAddLine(
		i_pOD := ADR(G_CANopen_CAN1.OD),(*Address of Object dictionary where index will be added*)
		i_Index := G_CANOPEN_ODINDEX_MF_DEVICE_NAME,
		i_ObjectCode := EPEC_CANopen.ObjectCode.OD_VAR,(*Type of index*)
		i_NumOfSubids := USINT#0,(*Number of subindexes*)
		i_TypeSpec := EPEC_CANopen.DataType.Deftype_STRING,(*Index datatype, either user defined or standard CiA 301*)
		i_ObjectAccess := G_CANOPEN_OD_ACCESS_NOWRITE OR G_CANOPEN_OD_ACCESS_SUB0NOWRITE,
		i_Sub0data := USINT#0,(*Value of subindex0 in array or (def)struct*)
		i_pIndexData := ADR(G_SystemInfo.DeviceName),
		i_itfSDOHandler := DWORD#0
	);
END_IF

(* 16#100A Manufacturer software version *)
IF G_CANopen_CAN1_VAR.OD_Error = EPEC_CANopen.Errors.NoError THEN
	G_CANopen_CAN1_VAR.OD_Error := CANopenODAddLine(
		i_pOD := ADR(G_CANopen_CAN1.OD),(*Address of Object dictionary where index will be added*)
		i_Index := G_CANOPEN_ODINDEX_MF_SW_VERSION,
		i_ObjectCode := EPEC_CANopen.ObjectCode.OD_VAR,(*Type of index*)
		i_NumOfSubids := USINT#0,(*Number of subindexes*)
		i_TypeSpec := EPEC_CANopen.DataType.Deftype_STRING,(*Index datatype, either user defined or standard CiA 301*)
		i_ObjectAccess := G_CANOPEN_OD_ACCESS_NOWRITE OR G_CANOPEN_OD_ACCESS_SUB0NOWRITE,
		i_Sub0data := USINT#0,(*Value of subindex0 in array or (def)struct*)
		i_pIndexData := ADR(G_SystemInfo.SWVersion),
		i_itfSDOHandler := DWORD#0
	);
END_IF

(* 16#1018   Vendor ID *)
IF G_CANopen_CAN1_VAR.OD_Error = EPEC_CANopen.Errors.NoError THEN
	G_CANopen_CAN1_VAR.OD_Error := CANopenODAddLine(
		i_pOD := ADR(G_CANopen_CAN1.OD),(*Address of Object dictionary where index will be added*)
		i_index := G_CANOPEN_ODINDEX_IDENTITY_OBJECT,
		i_ObjectCode := EPEC_CANopen.ObjectCode.OD_ARRAY, (*Type of index*)
		i_NumOfSubids := USINT#4,(*Number of subindexes*)
		i_TypeSpec := EPEC_CANopen.DataType.Deftype_UNSIGNED32,(*Index of 16-bit deftype*)
		i_ObjectAccess := G_CANOPEN_OD_ACCESS_NOWRITE OR G_CANOPEN_OD_ACCESS_SUB0NOWRITE,
		i_sub0data := USINT#4,(*Value of subindex0 in array or (def)struct*)
		i_pIndexData := ADR(G_SystemInfo.Identity),
		i_itfSDOHandler := DWORD#0
	);
END_IF
(* 16#2030   CodesysVersion *)
IF G_CANopen_CAN1_VAR.OD_Error = EPEC_CANopen.Errors.NoError THEN
	G_CANopen_CAN1_VAR.OD_Error := CANopenODAddLine(
		i_pOD := ADR(G_CANopen_CAN1.OD),(*Address of Object dictionary where index will be added*)
		i_index := 16#2030,
		i_ObjectCode := EPEC_CANopen.ObjectCode.OD_ARRAY, (*Type of index*)
		i_NumOfSubids := USINT#1,(*Number of subindexes*)
		i_TypeSpec := EPEC_CANopen.DataType.Deftype_UNSIGNED32,(*Index of 16-bit deftype*)
		i_ObjectAccess := G_CANOPEN_OD_ACCESS_NOWRITE OR G_CANOPEN_OD_ACCESS_SUB0NOWRITE,
		i_sub0data := USINT#1,(*Value of subindex0 in array or (def)struct*)
		i_pIndexData := ADR(G_SystemInfo.ToolsVersion),
		i_itfSDOHandler := DWORD#0
	);
END_IF

(* 16#2128 PDO Dummy Variable Index *)
IF G_CANopen_CAN1_VAR.OD_Error = EPEC_CANopen.Errors.NoError THEN
	G_CANopen_CAN1_VAR.OD_Error := CANopenODAddLine(
		i_pOD := ADR(G_CANopen_CAN1.OD),(*Address of Object dictionary where index will be added*)
		i_Index := 16#2128,
		i_ObjectCode := EPEC_CANopen.ObjectCode.OD_VAR,(*Type of index*)
		i_NumOfSubids := USINT#0,(*Number of subindexes*)
		i_TypeSpec := EPEC_CANopen.DataType.Deftype_UNSIGNED8,(*Index datatype, either user defined or standard CiA 301*)
		i_ObjectAccess := G_CANOPEN_OD_ACCESS_READWRITE,
		i_Sub0data := USINT#0,(*Value of subindex0 in array or (def)struct*)
		i_pIndexData := ADR(G_CAN1_VAR.TPDO_DUMMY),
		i_itfSDOHandler := DWORD#0
	);
END_IF

(* 16#2129 PDO Dummy Variable Index *)
IF G_CANopen_CAN1_VAR.OD_Error = EPEC_CANopen.Errors.NoError THEN
	G_CANopen_CAN1_VAR.OD_Error := CANopenODAddLine(
		i_pOD := ADR(G_CANopen_CAN1.OD),(*Address of Object dictionary where index will be added*)
		i_Index := 16#2129,
		i_ObjectCode := EPEC_CANopen.ObjectCode.OD_VAR,(*Type of index*)
		i_NumOfSubids := USINT#0,(*Number of subindexes*)
		i_TypeSpec := EPEC_CANopen.DataType.Deftype_UNSIGNED8,(*Index datatype, either user defined or standard CiA 301*)
		i_ObjectAccess := G_CANOPEN_OD_ACCESS_READWRITE,
		i_Sub0data := USINT#0,(*Value of subindex0 in array or (def)struct*)
		i_pIndexData := ADR(G_CAN1_VAR.RPDO_DUMMY),
		i_itfSDOHandler := DWORD#0
	);
END_IF

(* 16#2130   Application version *)
IF G_CANopen_CAN1_VAR.OD_Error = EPEC_CANopen.Errors.NoError THEN
	G_CANopen_CAN1_VAR.OD_Error := CANopenODAddLine(
		i_pOD := ADR(G_CANopen_CAN1.OD),(*Address of Object dictionary where index will be added*)
		i_index := 16#2130,
		i_ObjectCode := EPEC_CANopen.ObjectCode.OD_ARRAY, (*Type of index*)
		i_NumOfSubids := USINT#10,(*Number of subindexes*)
		i_TypeSpec := EPEC_CANopen.DataType.Deftype_STRING,(*Index of 16-bit deftype*)
		i_ObjectAccess := G_CANOPEN_OD_ACCESS_NOWRITE OR G_CANOPEN_OD_ACCESS_SUB0NOWRITE,
		i_sub0data := USINT#10,(*Value of subindex0 in array or (def)struct*)
		i_pIndexData := ADR(G_SystemInfo.SoftwareInformation),
		i_itfSDOHandler := DWORD#0
	);
END_IF

(* 16#2131 Parameter CSV unique ID *)
IF G_CANopen_CAN1_VAR.OD_Error = EPEC_CANopen.Errors.NoError THEN
	G_CANopen_CAN1_VAR.OD_Error := CANopenODAddLine(
		i_pOD := ADR(G_CANopen_CAN1.OD),(*Address of Object dictionary where index will be added*)
		i_Index := 16#2131,
		i_ObjectCode := EPEC_CANopen.ObjectCode.OD_VAR,(*Type of index*)
		i_NumOfSubids := USINT#0,(*Number of subindexes*)
		i_TypeSpec := EPEC_CANopen.DataType.Deftype_UNSIGNED16,(*Index datatype, either user defined or standard CiA 301*)
		i_ObjectAccess := G_CANOPEN_OD_ACCESS_NOWRITE OR G_CANOPEN_OD_ACCESS_SUB0NOWRITE,
		i_Sub0data := USINT#0,(*Value of subindex0 in array or (def)struct*)
		i_pIndexData := ADR(G_CAN1_VAR.Parameter_CSV_unique_ID),
		i_itfSDOHandler := DWORD#0
	);
END_IF

(* 16#2150   CODESYS communication enabled *)
IF G_CANopen_CAN1_VAR.OD_Error = EPEC_CANopen.Errors.NoError THEN
	G_CANopen_CAN1_VAR.OD_Error := CANopenODAddLine(
		i_pOD := ADR(G_CANopen_CAN1.OD),(*Address of Object dictionary where index will be added*)
		i_index := 16#2150,
		i_ObjectCode := EPEC_CANopen.ObjectCode.OD_ARRAY, (*Type of index*)
		i_NumOfSubids := USINT#10,(*Number of subindexes*)
		i_TypeSpec := EPEC_CANopen.DataType.Deftype_UNSIGNED16,(*Index of 16-bit deftype*)
		i_ObjectAccess := G_CANOPEN_OD_ACCESS_READWRITE OR G_CANOPEN_OD_ACCESS_SUB0NOWRITE,
		i_sub0data := USINT#10,(*Value of subindex0 in array or (def)struct*)
		i_pIndexData := ADR(G_SystemInfo.CAN1_Comms),
		i_itfSDOHandler := DWORD#0
	);
END_IF

(* 16#2151   CODESYS communication enabled *)
IF G_CANopen_CAN1_VAR.OD_Error = EPEC_CANopen.Errors.NoError THEN
	G_CANopen_CAN1_VAR.OD_Error := CANopenODAddLine(
		i_pOD := ADR(G_CANopen_CAN1.OD),(*Address of Object dictionary where index will be added*)
		i_index := 16#2151,
		i_ObjectCode := EPEC_CANopen.ObjectCode.OD_ARRAY, (*Type of index*)
		i_NumOfSubids := USINT#10,(*Number of subindexes*)
		i_TypeSpec := EPEC_CANopen.DataType.Deftype_UNSIGNED16,(*Index of 16-bit deftype*)
		i_ObjectAccess := G_CANOPEN_OD_ACCESS_READWRITE OR G_CANOPEN_OD_ACCESS_SUB0NOWRITE,
		i_sub0data := USINT#10,(*Value of subindex0 in array or (def)struct*)
		i_pIndexData := ADR(G_SystemInfo.CAN2_Comms),
		i_itfSDOHandler := DWORD#0
	);
END_IF

(*16#2170 Application log error count *)
IF G_CANopen_CAN1_VAR.OD_Error = EPEC_CANopen.Errors.NoError THEN
	G_CANopen_CAN1_VAR.OD_Error := CANopenODAddLine(
		i_pOD:= ADR(G_CANopen_CAN1.OD), (*Address of Object dictionary where index will be added *)
		i_index:= 16#2170,
		i_ObjectCode:= EPEC_CANopen.ObjectCode.OD_VAR, (*Type of index*)
		i_NumOfSubids:= USINT#0,(*Number of subindexes*)
		i_TypeSpec:= EPEC_CANopen.DataType.Deftype_UNSIGNED32,(*Index of 32 - bit deftype *)
		i_ObjectAccess:= G_CANOPEN_OD_ACCESS_NOWRITE OR G_CANOPEN_OD_ACCESS_SUB0NOWRITE,
		i_sub0data := USINT#0,(*Value of subindex0 in array or (def)struct*)
		i_pIndexData:= ADR(G_Logs.ApplicationLog.count),
		i_itfSDOHandler:= DWORD#0
	);
END_IF

(*16#2171 Application log domain *)
	IF G_CANopen_CAN1_VAR.OD_Error = EPEC_CANopen.Errors.NoError THEN
	G_CANopen_CAN1.AppLogDomain.DataSize:= SIZEOF(G_Logs.ApplicationLog.loglines) * 8;
	G_CANopen_CAN1.AppLogDomain.pData:= ADR(G_Logs.ApplicationLog.loglines);

	G_CANopen_CAN1_VAR.OD_Error := CANopenODAddLine(
		i_pOD:= ADR(G_CANopen_CAN1.OD), (*Address of Object dictionary where index will be added *)
		i_index:= 16#2171,
		i_ObjectCode:= EPEC_CANOPEN.ObjectCode.OD_DOMAIN, (*Type of index*)
		i_NumOfSubids:= USINT#0,(*Number of subindexes*)
		i_TypeSpec:= EPEC_CANOPEN.DataType.Deftype_Domain,(*Domain deftype *)
		i_ObjectAccess:= G_CANOPEN_OD_ACCESS_NOWRITE,
		i_sub0data:= USINT#0,(*Value of subindex0 in array or (def)struct*)
		i_pIndexData:= ADR(G_CANopen_CAN1.AppLogDomain),
		i_itfSDOHandler:= DWORD#0
	);
END_IF

          
END_PROGRAM

(* NOTE! NOTE! NOTE! NOTE! NOTE! NOTE! NOTE! NOTE! NOTE! NOTE! NOTE! This object is created by Epec MultiTool User changes are overwritten when project is imported Content - CANopen data update This PRG contains non safety-related code. The following attribute is autogenerated. Do not remove. *)
{attribute 'location' := '16#800'}
PROGRAM Handle_CANopen_CAN1
  VAR_OUTPUT
    o_Error : BOOL := FALSE;
  END_VAR

            (* Update callback data *)
IF G_CAN.Channel1.GetLatestError() <> DWORD#0 THEN
	G_CANopen_CAN1_VAR.Callback_Error := EPEC_CANopen.Errors.CallbackError;
ELSE
	G_CANopen_CAN1_VAR.Callback_Error := EPEC_CANopen.Errors.NoError;
END_IF

(* Update protocol data *)
G_CANopen_CAN1.HB_Handler.Update(
	i_Enable := TRUE,
	o_Error => G_CANopen_CAN1_VAR.HB_Error
);
G_CANopen_CAN1.NMT_Handler.Update(
	i_Enable := TRUE,
	o_Error => G_CANopen_CAN1_VAR.NMT_Error
);
G_CANopen_CAN1.SSDO_Handler.Update(
	i_Enable := TRUE,
	o_Error => G_CANopen_CAN1_VAR.SSDO_Error
);
G_CANopen_CAN1.GFC_Handler.Update(
	i_Enable := TRUE,
	o_Error => G_CANopen_CAN1_VAR.GFC_Error
);

IF G_CANopen_CAN1_VAR.HB_Error = EPEC_CANopen.Errors.NoError AND
	G_CANopen_CAN1_VAR.NMT_Error = EPEC_CANopen.Errors.NoError AND
	G_CANopen_CAN1_VAR.SSDO_Error = EPEC_CANopen.Errors.NoError AND
	G_CANopen_CAN1_VAR.GFC_Error = EPEC_CANopen.Errors.NoError
THEN
	o_Error := FALSE;
ELSE
	o_Error := TRUE;

	EPEC_SERRLOG.S_AddError_DWORD(i_ErrorCode:= ApplicationErrors.CANOPEN_UPDATE_HB, i_LibraryErrorCode:= INT_TO_DINT(G_CANopen_CAN1_VAR.HB_Error), i_Info1:= 0, i_Info2:= 1);
	EPEC_SERRLOG.S_AddError_DWORD(i_ErrorCode:= ApplicationErrors.CANOPEN_UPDATE_NMT, i_LibraryErrorCode:= INT_TO_DINT(G_CANopen_CAN1_VAR.NMT_Error), i_Info1:= 0, i_Info2:= 1);
	EPEC_SERRLOG.S_AddError_DWORD(i_ErrorCode:= ApplicationErrors.CANOPEN_UPDATE_SSDO, i_LibraryErrorCode:= INT_TO_DINT(G_CANopen_CAN1_VAR.SSDO_Error), i_Info1:= 0, i_Info2:= 1);
	EPEC_SERRLOG.S_AddError_DWORD(i_ErrorCode:= ApplicationErrors.CANOPEN_UPDATE_GFC, i_LibraryErrorCode:= INT_TO_DINT(G_CANopen_CAN1_VAR.GFC_Error), i_Info1:= 0, i_Info2:= 1);

END_IF

(*Check for NMT reset *)
IF G_CANopen_CAN1.NMT.StateChanged THEN
	IF G_CANopen_CAN1.NMT.LastNmtCommand = EPEC_CANopen.NMTCommand.Reset OR
		G_CANopen_CAN1.NMT.LastNmtCommand = EPEC_CANopen.NMTCommand.ResetCommunication
	THEN
		(* If there is an NMT reset command for the IEC application CANopen device,
		   This is only informative, application decides how to react to the command *)
		G_StatusFlags.CANopenCan1NMTResetRequest := TRUE;
	END_IF
END_IF


          
END_PROGRAM

(* NOTE! NOTE! NOTE! NOTE! NOTE! NOTE! NOTE! NOTE! NOTE! NOTE! NOTE! This object is created by Epec MultiTool User changes are overwritten when project is imported Content - Init IO. This PRG contains safety-related code. The following attribute is autogenerated. Do not remove. *)
PROGRAM Init_IO
  VAR_OUTPUT
    o_Ready : SAFEBOOL := FALSE;
    o_Error : BOOL := FALSE;
    o_ErrorInConnector : DWORD := DWORD#0;
    o_ErrorInPin : DWORD := DWORD#0;
    o_FWErrorCode : EPEC_SYSTEM.SYSTEM_ERROR_CODES;
  END_VAR
  VAR
    result : EPEC_SYSTEM.SYSTEM_ERROR_CODES;
    pin : DWORD := DWORD#0;
    connector : DWORD := DWORD#0;
    info1 : DWORD := DWORD#0;  (* MSW connector, LSW pin *)
    info2 : DWORD := DWORD#0;  (* error specific *)
  END_VAR

            IF result = EPEC_SYSTEM.SYSTEM_ERROR_CODES.FW_ERR_OK THEN
	result := EPEC_IODRV.IoDrvSetState(EPEC_IODRV.IoDrvStates.IODRV_STATE_CONFIGURATION);
END_IF

IF result = EPEC_SYSTEM.SYSTEM_ERROR_CODES.FW_ERR_OK THEN
	connector := 255; // internal
	pin := 1;
	result := EPEC_IODRV.IoDrvAISetMode(EPEC_HW.IO_Channels.PIN_INT_AI_PWR_SWT_AFTER, EPEC_IODRV.IoDrvModes.IODRV_MODE_AI_ENABLED);
END_IF

IF result = EPEC_SYSTEM.SYSTEM_ERROR_CODES.FW_ERR_OK THEN
	pin := 2;
	result := EPEC_IODRV.IoDrvAISetMode(EPEC_HW.IO_Channels.PIN_INT_AI_PWR_SWT_BEFORE, EPEC_IODRV.IoDrvModes.IODRV_MODE_AI_ENABLED);
END_IF

IF result = EPEC_SYSTEM.SYSTEM_ERROR_CODES.FW_ERR_OK THEN
	pin := 3;
	result := EPEC_IODRV.IoDrvAISetMode(EPEC_HW.IO_Channels.PIN_INT_AI_REF_VOLTAGE, EPEC_IODRV.IoDrvModes.IODRV_MODE_AI_ENABLED);
END_IF

IF result = EPEC_SYSTEM.SYSTEM_ERROR_CODES.FW_ERR_OK THEN
	pin := 4;
	result := EPEC_IODRV.IoDrvDOSetConfig(EPEC_HW.IO_Channels.PIN_INT_DO_REF_VOLTAGE_10V, NOT(G_CONSTANTS.DIAG_REF_TYPE_5V));
END_IF

IF result = EPEC_SYSTEM.SYSTEM_ERROR_CODES.FW_ERR_OK THEN
	pin := 5;
	result := EPEC_IODRV.IoDrvAISetMode(EPEC_HW.IO_Channels.PIN_INT_AI_TEMP1, EPEC_IODRV.IoDrvModes.IODRV_MODE_AI_ENABLED);
END_IF

IF result = EPEC_SYSTEM.SYSTEM_ERROR_CODES.FW_ERR_OK THEN
	pin := 6;
	result := EPEC_IODRV.IoDrvAISetMode(EPEC_HW.IO_Channels.PIN_INT_AI_TEMP2, EPEC_IODRV.IoDrvModes.IODRV_MODE_AI_ENABLED);
END_IF

IF result = EPEC_SYSTEM.SYSTEM_ERROR_CODES.FW_ERR_OK THEN
	pin := 7;
	result := EPEC_IODRV.IoDrvAISetMode(EPEC_HW.IO_Channels.PIN_INT_AI_VIn_1_1, EPEC_IODRV.IoDrvModes.IODRV_MODE_AI_ENABLED);
END_IF

IF result = EPEC_SYSTEM.SYSTEM_ERROR_CODES.FW_ERR_OK THEN
	pin := 8;
	result := EPEC_IODRV.IoDrvAISetMode(EPEC_HW.IO_Channels.PIN_INT_AI_VIN_POWER, EPEC_IODRV.IoDrvModes.IODRV_MODE_AI_ENABLED);
END_IF

IF result = EPEC_SYSTEM.SYSTEM_ERROR_CODES.FW_ERR_OK THEN
	pin := 9;
	result := EPEC_IODRV.IoDrvAISetMode(EPEC_HW.IO_Channels.PIN_INT_AI_MCU_TEMP, EPEC_IODRV.IoDrvModes.IODRV_MODE_AI_ENABLED);
END_IF

IF result = EPEC_SYSTEM.SYSTEM_ERROR_CODES.FW_ERR_OK THEN
	pin := 10;
	result := EPEC_IODRV.IoDrvAISetMode(EPEC_HW.IO_Channels.PIN_INT_AI_5VAN, EPEC_IODRV.IoDrvModes.IODRV_MODE_AI_ENABLED);
END_IF

IF result = EPEC_SYSTEM.SYSTEM_ERROR_CODES.FW_ERR_OK THEN
	pin := 11;
	result := EPEC_IODRV.IoDrvAISetMode(EPEC_HW.IO_Channels.PIN_INT_AI_SBC_TEMP, EPEC_IODRV.IoDrvModes.IODRV_MODE_AI_ENABLED);
END_IF
  
IF result = EPEC_SYSTEM.SYSTEM_ERROR_CODES.FW_ERR_OK THEN
	result := EPEC_IODRV.IoDrvSetState(EPEC_IODRV.IoDrvStates.IODRV_STATE_RUN);
	o_FWErrorCode := result;
END_IF

IF result <> EPEC_SYSTEM.SYSTEM_ERROR_CODES.FW_ERR_OK THEN
	o_Error:=TRUE;
	o_ErrorInConnector := connector;
	o_ErrorInPin := pin;
	o_FWErrorCode := result;

	info1:= SHL(connector, 16) OR pin;
	EPEC_SERRLOG.S_AddError_DWORD(
		i_ErrorCode:= ApplicationErrors.IO_INIT,
		i_LibraryErrorCode:= result,
		i_Info1:= info1, // MSW connector, LSW pin
		i_Info2:= info2 // error specific
	);
END_IF

o_Ready:=TRUE;

          
END_PROGRAM

(* NOTE! NOTE! NOTE! NOTE! NOTE! NOTE! NOTE! NOTE! NOTE! NOTE! NOTE! This object is created by Epec MultiTool User changes are overwritten when project is imported Content: - Input pin data update. This PRG contains non safety-related code. The following attribute is autogenerated. Do not remove. *)
{attribute 'hide_all_locals'}
{attribute 'location' := '16#800'}
PROGRAM Inputs
  VAR_INPUT
    i_Enable : BOOL := TRUE;
    i_Initialize : BOOL := TRUE;
  END_VAR
  VAR_OUTPUT
    o_InitReady : BOOL := FALSE;
    o_AI_POWER1_SUPPLY_Diagnostic : DWORD;  (* Measurent for power switch input voltage [unscaled] *)
    o_AI_POWER1_OUTPUT_Diagnostic : DWORD;  (* Measurement for power switch output voltage [unscaled]. *)
    o_AI_REF_OUTPUT_MAIN_Diagnostic : DWORD;  (* Measurement for selectable reference voltage (5/10V) [unscaled]. *)
    o_TEMP_PCB_MAIN_Diagnostic : DWORD;  (* Measurement for PCB temperature 1 [unscaled] *)
    o_TEMP_PCB_RED_Diagnostic : DWORD;  (* Measurement for PCB temperature 2 [unscaled] *)
    o_VIN_1_1_Diagnostic : DWORD;  (* Measurement for supply pin voltage [unscaled] *)
    o_VIN_POWER_Diagnostic : DWORD;  (* Measurement for Vin power [unscaled] *)
    o_TEMP_MCU_Diagnostic : DINT;  (* Measurement for MCU temperature [0.1C] *)
    o_AI_5VAN_Diagnostic : DWORD;  (* Measurement for 5VAN voltage [unscaled] *)
    o_AI_SBC_TEMP_Diagnostic : DINT;  (* SBC temperature [0.1 C] *)
  END_VAR
  VAR
    AI_POWER1_SUPPLY_Diagnostic : DWORD;  (* Measurent for power switch input voltage (Mapped variable) *)
    AI_POWER1_OUTPUT_Diagnostic : DWORD;  (* Measurement for power switch output voltage (Mapped variable).. *)
    AI_REF_OUTPUT_MAIN_Diagnostic : DWORD;  (* Measurement for selectable reference voltage (5/10V). (Mapped variable) *)
    TEMP_PCB_MAIN_Diagnostic : DWORD;  (* Measurement for PCB temperature 1 (Mapped variable) *)
    TEMP_PCB_RED_Diagnostic : DWORD;  (* Measurement for PCB temperature 2 (Mapped variable) *)
    VIN_1_1_Diagnostic : DWORD;  (* Measurement for supply pin voltage (Mapped variable) *)
    VIN_POWER_Diagnostic : DWORD;  (* Measurement for Vin power (Mapped variable) *)
    TEMP_MCU_Diagnostic : DINT;  (* Measurement for MCU temperature (Mapped variable) *)
    AI_5VAN_Diagnostic : DWORD;  (* Measurement for 5VAN voltage (Mapped variable) *)
    AI_SBC_TEMP_Diagnostic : DINT;  (* SBC temperature [0.1 C] *)
  END_VAR

            IF(i_Initialize) THEN
	o_InitReady:= TRUE;
  
ELSE

	(* Copy measured diagnostic signals to outputs *)
	o_AI_POWER1_SUPPLY_Diagnostic := AI_POWER1_SUPPLY_Diagnostic;
	o_AI_POWER1_OUTPUT_Diagnostic := AI_POWER1_OUTPUT_Diagnostic;
	o_AI_REF_OUTPUT_MAIN_Diagnostic := AI_REF_OUTPUT_MAIN_Diagnostic;
	o_TEMP_PCB_MAIN_Diagnostic := TEMP_PCB_MAIN_Diagnostic;
	o_TEMP_PCB_RED_Diagnostic := TEMP_PCB_RED_Diagnostic;
	o_VIN_1_1_Diagnostic := VIN_1_1_Diagnostic;
	o_VIN_POWER_Diagnostic := VIN_POWER_Diagnostic;
	o_TEMP_MCU_Diagnostic := TEMP_MCU_Diagnostic;
	o_AI_5VAN_Diagnostic := AI_5VAN_Diagnostic;
	o_AI_SBC_TEMP_Diagnostic := AI_SBC_TEMP_Diagnostic;


  
END_IF

          
END_PROGRAM
